FUNCTION F_astroRad2Hms : LREAL
VAR_INPUT
	hh:	LREAL;	// angle in radians
END_VAR
VAR
	value:		LREAL;
	hours:		INT;
	minutes:	INT;
	seconds:	LREAL;
	
	sign:	int := 1;
END_VAR

IF hh < 0.0 THEN
	sign	:= -1;
	hh		:= -hh;
END_IF

value := hh / GCL.C_2PI * 24.0; 	// rad to hours


hours	:= TRUNC_INT(value);
minutes := TRUNC_INT((value - hours)*60.0);
seconds := (value - hours - minutes/60.0)*3600.0;

hours	:= hours * sign;	// put back the sign

					
F_astroRad2Hms	:= hours * 10000 + minutes * 100 + seconds;

END_FUNCTION

(* stored: Version 1.1.0.1, ProductVersion 3.1.4022.9
   POU F_astroRad2Hms: Id {72247f6a-c059-41d6-802f-ffdd182b0698}, SpecialFunc None *)
